{attribute 'linkalways'} 
{attribute 'no_explicit_call' := 'This FB is a CLASS and must be accessed using methods or properties'}
{attribute 'enable_dynamic_creation'}
FUNCTION_BLOCK _ETcVnRectangleIntersection EXTENDS EnumDatatypeBase
VAR
	localData : ETcVnRectangleIntersection;
	activeData : REFERENCE TO ETcVnRectangleIntersection;
	enumBaseDatatype : _DINT(localData);
END_VAR

METHOD PRIVATE AddLocalEnumeration
VAR_INPUT
	Enumeration : T_MAXSTRING;
	Value : ETcVnRectangleIntersection;
END_VAR
AddEnumeration(Enumeration, Value);
END_METHOD

PROPERTY PUBLIC Address : PVOID
GET
Address := ADR(activeData);
END_GET
END_PROPERTY

METHOD PUBLIC ClearReference
VAR_INPUT
END_VAR
activeData REF= localData;
SetBaseDatatypeReference();
END_METHOD

METHOD PUBLIC Clone : I_Datatype
VAR
    pClone : POINTER TO _ETcVnRectangleIntersection;
END_VAR
pClone := __NEW(_ETcVnRectangleIntersection(InitialValue := Value));
Clone := pClone^;
END_METHOD

METHOD FB_init : BOOL
VAR_INPUT
	bInitRetains : BOOL; // if TRUE, the retain variables are initialized (warm start / cold start)
	bInCopyCode : BOOL;  // if TRUE, the instance afterwards gets moved into the copy code (online change)
	InitialValue : ETcVnRectangleIntersection;
END_VAR
localData := InitialValue;
AddBaseDatatype(enumBaseDatatype);
ClearReference();

AddLocalEnumeration('TCVN_RI_NONE', ETcVnRectangleIntersection.TCVN_RI_NONE);
AddLocalEnumeration('TCVN_RI_PARTIAL', ETcVnRectangleIntersection.TCVN_RI_PARTIAL);
AddLocalEnumeration('TCVN_RI_FULL', ETcVnRectangleIntersection.TCVN_RI_FULL);
END_METHOD

PROPERTY PUBLIC Identifier : T_MAXSTRING
GET
Identifier := 'ETcVnRectangleIntersection';
END_GET
END_PROPERTY

METHOD IsEnumeratorValueEqual : BOOL
VAR_INPUT
	Enumerator : I_KeyValueForwardEnumerator;
END_VAR
VAR
	storedValue : ETcVnRectangleIntersection;
END_VAR
IF NOT Enumerator.TryGet(storedValue) THEN
	RETURN;
END_IF

IsEnumeratorValueEqual := storedValue = activeData;
END_METHOD

METHOD PUBLIC MakeReferenceTo
VAR_INPUT
	ReferenceTarget : REFERENCE TO ETcVnRectangleIntersection;
END_VAR
activeData REF= ReferenceTarget;
SetBaseDatatypeReference();
END_METHOD

METHOD PROTECTED SetBaseDatatypeReference
VAR_INPUT
END_VAR
enumBaseDatatype.MakeReferenceTo(activeData);
END_METHOD

PROPERTY PUBLIC Size : UDINT
GET
Size := SIZEOF(activeData);
END_GET
END_PROPERTY

METHOD TryMakeReferenceTo : BOOL
VAR_INPUT
	Target : I_Datatype;
END_VAR
VAR
	targetAsEnum : I_EnumDatatype;
	pTargetData : POINTER TO ETcVnRectangleIntersection;
END_VAR
IF NOT Target.TryResolveAsEnumDatatype(targetAsEnum) THEN
	RETURN;
END_IF

IF targetAsEnum.Identifier <> Identifier THEN
	RETURN;
END_IF

pTargetData := Target.Address;
activeData REF= pTargetData^;
SetBaseDatatypeReference();
TryMakeReferenceTo := TRUE;
END_METHOD

PROPERTY PUBLIC Value : ETcVnRectangleIntersection
GET
Value := activeData;
END_GET
SET
activeData := Value;
END_SET
END_PROPERTY

END_FUNCTION_BLOCK

(* stored: Version 1.1.0.1
   POU _ETcVnRectangleIntersection: Id {4d86df11-16a6-47d5-b5f7-14399101d9a9}, SpecialFunc None
   Folder Constructor: Id {ba2fb915-48dc-48bb-83cb-37896ab9d7e5}
   Folder Private: Id {24953008-7e17-4540-9971-dff733644c94}
   Folder Protected: Id {1499d659-d045-4a7a-add0-6187ce872e7f}
   Method AddLocalEnumeration: Id {9199f45d-04b4-4c81-a958-91c1cdf27db1}
   Property Address: Id {d542029a-2d93-4c4c-860e-b744ddcec805}
   Get Get: Id {cedca429-4861-4a49-ac10-248a3a8d81d7}
   Method ClearReference: Id {92b0bdd1-05aa-4227-bdd3-ab2627a4640b}
   Method Clone: Id {c6aacbd3-ff19-4972-bec8-20f0f8ef24f2}
   Method FB_init: Id {f76cb8d9-cb42-4797-b6dc-96fd3bfe5f1d}
   Property Identifier: Id {dd79172a-022d-4541-b57e-3355fce9b857}
   Get Get: Id {254cf817-e855-403f-8e16-8d1e9375ba19}
   Method IsEnumeratorValueEqual: Id {fb34ee3a-ddb9-492c-b536-a4673f917657}
   Method MakeReferenceTo: Id {d484a754-dff7-4618-93d2-d3b4be7ce111}
   Method SetBaseDatatypeReference: Id {939ccb5b-36d3-451c-bd6e-93395535c150}
   Property Size: Id {9519ead7-2cf4-4b0a-9a6a-a962869fb80d}
   Get Get: Id {cccbf82d-6669-41c0-b897-c7ad01e6fca8}
   Method TryMakeReferenceTo: Id {c93f7dd9-06ac-4f48-9b55-5525401293c9}
   Property Value: Id {1037057b-d1c1-47d4-8818-187a6f835eb3}
   Get Get: Id {c575a351-3b0c-4c68-9ca3-1233f527af15}
   Set Set: Id {84048b88-8e43-4526-bbe6-99a9e0c871b7} *)
